TYPE ST_EL6633 :
STRUCT
	
	// TERMINAL - EL66633	Profinet Protocol	 (Term 12)
	sTerminalName                                           :   STRING(200):= 'EL6633 | Profinet Protocol';
	stTerminalInfo											: 	ST_Terminal_Info;

END_STRUCT
END_TYPE

(* stored: Version 1.1.0.1, ProductVersion 3.1.4024.13
   DUT ST_EL6633: Id {98f9bc9d-d8a8-480d-9373-00c6fa321ef2} *)
